// TIA Portal project "Proporcional" (V15)

(* hardware
DEVICE "S7-1200 station_1"  S7-1200 Station
   slot 0: "Rack_0"  S7-1200 Rack  Rack  V1.0
   slot 1: "PLC_1"  CPU 1214C DC/DC/DC  6ES7 214-1AG40-0XB0  V4.2
   slot 3: "AQ 1x12BIT_1"  AQ1 signal board  6ES7 232-4HA30-0XB0  V1.0
*)

// ===== PLC "PLC_1"  CPU 1214C DC/DC/DC =====

VAR_GLOBAL   // PLC tag table "Tabla de variables estándar"
   "Tag_1" AT %IW64 : Int;
   "Tag_2" AT %QW80 : Int;
   "Tag_3" AT %MD10 : DInt;
   "Calefactor" AT %Q0.0 : Bool;
END_VAR

DATA_BLOCK "Mis_datos"   // DB1
{ S7_Optimized_Access := 'TRUE' }
VERSION : 0.1
   VAR
      Temperatura : Real;
      SP : Real;
      Error : Real;
      Error_Porce : Real;
      EFC_Porce : Real;
      Tiempo : Real;
      SP_Porce : Real;
      Ganancia : Real;
      TON : Real;
      Intercepto : Real;
   END_VAR
BEGIN
END_DATA_BLOCK

// folder: System blocks/Program resources

DATA_BLOCK "Temporizador"   // DB2
{ S7_Optimized_Access := 'TRUE' }
AUTHOR : Simatic
FAMILY : IEC
NAME : IEC_TMR
VERSION : 1.0
// stored: InstanceOfName IEC_TIMER
"IEC_TIMER"
BEGIN
END_DATA_BLOCK

// folder: (top level)

FUNCTION "Acondicionamiento" : Void   // FC1, LAD
{ S7_Optimized_Access := 'TRUE' }
VERSION : 0.1
   VAR_TEMP
      Dato1 : Real;
      Dato2 : Real;
   END_VAR
BEGIN

REGION Network 1
   // Escalizar Temperatura
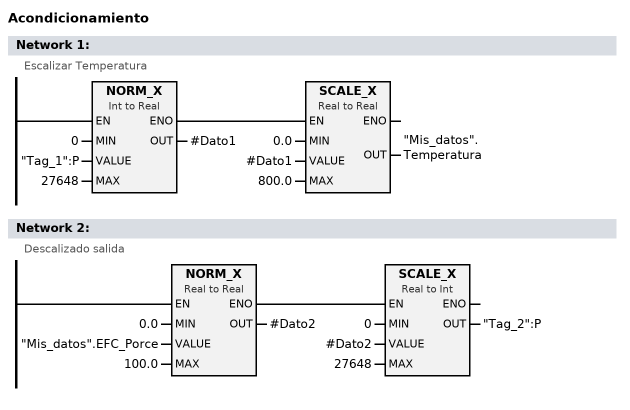
   RUNG wire#powerrail
      { S7_Templates := "[SrcType := Int, DestType := Real]" } Normalize(min := 0, value := "Tag_1":P, max := 27648, out => #Dato1)
      { S7_Templates := "[SrcType := Real, DestType := Real]" } Scale(min := 0.0, value := #Dato1, max := 800.0, out => "Mis_datos".Temperatura)
   END_RUNG
   // the same network as SCL:
   #Dato1 := NORM_X(MIN := 0, VALUE := "Tag_1":P, MAX := 27648);
   "Mis_datos".Temperatura := SCALE_X(MIN := 0.0, VALUE := #Dato1, MAX := 800.0);
END_REGION

REGION Network 2
   // Descalizado salida
   RUNG wire#powerrail
      { S7_Templates := "[SrcType := Real, DestType := Real]" } Normalize(min := 0.0, value := "Mis_datos".EFC_Porce, max := 100.0, out => #Dato2)
      { S7_Templates := "[SrcType := Real, DestType := Int]" } Scale(min := 0, value := #Dato2, max := 27648, out => "Tag_2":P)
   END_RUNG
   // the same network as SCL:
   #Dato2 := NORM_X(MIN := 0.0, VALUE := "Mis_datos".EFC_Porce, MAX := 100.0);
   "Tag_2":P := SCALE_X(MIN := 0, VALUE := #Dato2, MAX := 27648);
END_REGION
END_FUNCTION

FUNCTION "Proporcional" : Void   // FC2, LAD
{ S7_Optimized_Access := 'TRUE' }
VERSION : 0.1
   VAR_TEMP
      Dato3 : Real;
      Dato4 : Real;
   END_VAR
BEGIN

REGION Network 1
   // Hallar el error
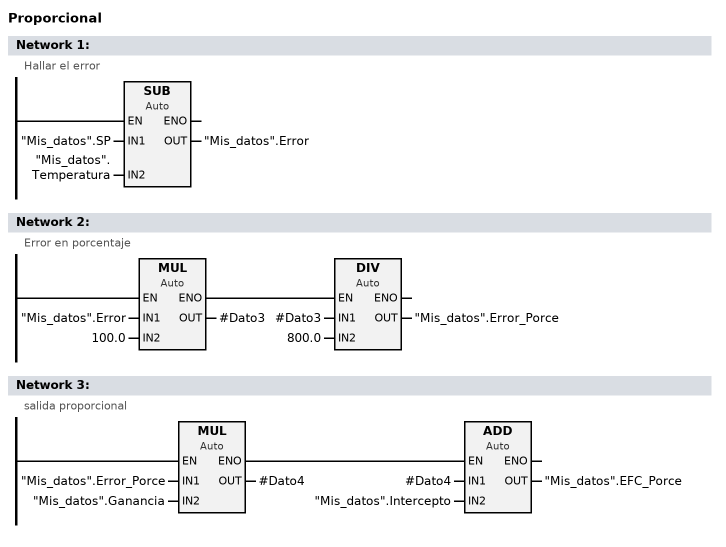
   RUNG wire#powerrail
      Sub(in1 := "Mis_datos".SP, in2 := "Mis_datos".Temperatura, out => "Mis_datos".Error)
   END_RUNG
   // the same network as SCL:
   "Mis_datos".Error := "Mis_datos".SP - "Mis_datos".Temperatura;
END_REGION

REGION Network 2
   // Error en porcentaje
   RUNG wire#powerrail
      Mul(in1 := "Mis_datos".Error, in2 := 100.0, out => #Dato3)
      Div(in1 := #Dato3, in2 := 800.0, out => "Mis_datos".Error_Porce)
   END_RUNG
   // the same network as SCL:
   #Dato3 := "Mis_datos".Error * 100.0;
   "Mis_datos".Error_Porce := #Dato3 / 800.0;
END_REGION

REGION Network 3
   // salida proporcional
   RUNG wire#powerrail
      Mul(in1 := "Mis_datos".Error_Porce, in2 := "Mis_datos".Ganancia, out => #Dato4)
      Add(in1 := #Dato4, in2 := "Mis_datos".Intercepto, out => "Mis_datos".EFC_Porce)
   END_RUNG
   // the same network as SCL:
   #Dato4 := "Mis_datos".Error_Porce * "Mis_datos".Ganancia;
   "Mis_datos".EFC_Porce := #Dato4 + "Mis_datos".Intercepto;
END_REGION
END_FUNCTION

FUNCTION "PWM" : Void   // FC3, LAD
{ S7_Optimized_Access := 'TRUE' }
VERSION : 0.1
   VAR_TEMP
      Dato5 : Real;
   END_VAR
BEGIN

REGION Network 1
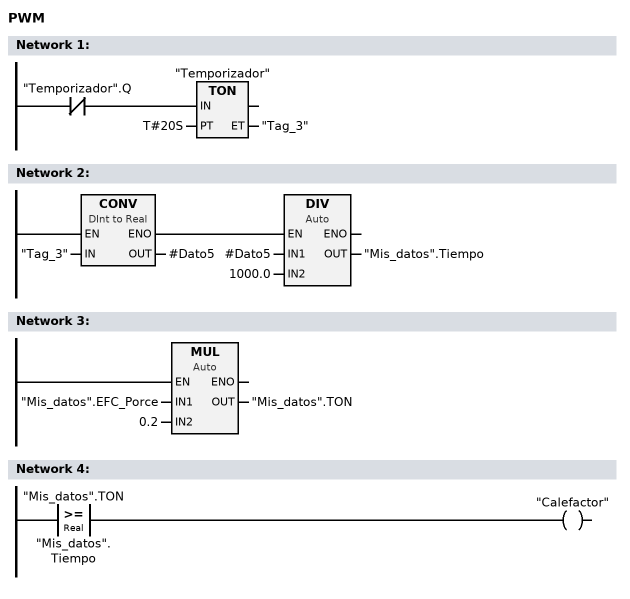
   "Temporizador".TON(IN := NOT "Temporizador".Q, PT := T#20S, ET => "Tag_3");
END_REGION

REGION Network 2
   RUNG wire#powerrail
      { S7_Templates := "[SrcType := DInt, DestType := Real]" } Convert(in := "Tag_3", out => #Dato5)
      Div(in1 := #Dato5, in2 := 1000.0, out => "Mis_datos".Tiempo)
   END_RUNG
   // the same network as SCL:
   #Dato5 := DINT_TO_REAL("Tag_3");
   "Mis_datos".Tiempo := #Dato5 / 1000.0;
END_REGION

REGION Network 3
   RUNG wire#powerrail
      Mul(in1 := "Mis_datos".EFC_Porce, in2 := 0.2, out => "Mis_datos".TON)
   END_RUNG
   // the same network as SCL:
   "Mis_datos".TON := "Mis_datos".EFC_Porce * 0.2;
END_REGION

REGION Network 4
   RUNG wire#powerrail
      { S7_Templates := "SrcType := Real" } GE_Contact(in1 := "Mis_datos".TON, in2 := "Mis_datos".Tiempo)
      Coil( "Calefactor" )
   END_RUNG
   // the same network as SCL:
   "Calefactor" := "Mis_datos".TON >= "Mis_datos".Tiempo;
END_REGION
END_FUNCTION

ORGANIZATION_BLOCK "Main"   // OB1, LAD, ProgramCycle
TITLE = "Main Program Sweep (Cycle)"
{ S7_Optimized_Access := 'TRUE' }
VERSION : 0.1
   VAR_INPUT
      Initial_Call : Bool;   // Initial call of this OB
      Remanence : Bool;   // =True, if remanent data are available
   END_VAR
BEGIN

REGION Network 1
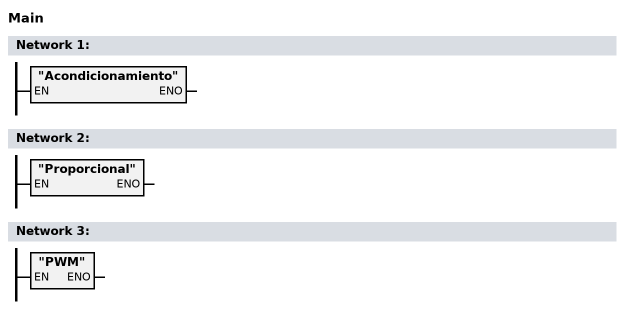
   RUNG wire#powerrail
      "Acondicionamiento"()
   END_RUNG
   // the same network as SCL:
   "Acondicionamiento"();
END_REGION

REGION Network 2
   RUNG wire#powerrail
      "Proporcional"()
   END_RUNG
   // the same network as SCL:
   "Proporcional"();
END_REGION

REGION Network 3
   RUNG wire#powerrail
      "PWM"()
   END_RUNG
   // the same network as SCL:
   "PWM"();
END_REGION
END_ORGANIZATION_BLOCK